TYPE StrMessage_t : String(255); END_TYPE

(* stored: Version 1.1.0.1, ProductVersion 3.1.4024.12
   DUT StrMessage_t: Id {87a84b72-d28f-4fcd-b96a-7652948c04c6} *)
